// TIA Portal V20 export
DATA_BLOCK "EmData"   // DB92
// stored: Access Published, MemoryReserve 100, Namespace Unit1
   VAR
      anodeElectrode : DInt;
      cathodeElectrode : DInt;
      currentTotalElectrode : DInt;
      targetTotalElectrode : DInt := 39;
      oldTotalElectrode : DInt;
      remainValue : DInt;   // Return reminder of divison.
      cpm : DInt := 80;
      homing : Bool;
      ReelCutStackCellCount : LReal;
      PartData : Struct
         EM4 : "LER_typePartDataEm4";
         EM5 : "LER_typePartDataEm5";
         EM6 : "LER_typePartDataEm6";
         EM7 : "LER_typePartDataEm7";
         clearPartData : "LER_typePartData";
         clearTableBuffer : Array[0..59] of "LER_typeUnitData";
      END_STRUCT;
      calculateResult : Struct
         sepaClampCutterAxisX { S7_SetPoint := 'True'} : "LBC_typeAxis64PosConfiguration";
         sepaClampCutterAxisZ { S7_SetPoint := 'True'} : "LBC_typeAxis64PosConfiguration";
         sepaGripperAxisX { S7_SetPoint := 'True'} : "LBC_typeAxis64PosConfiguration";
         pusherAxisZ { S7_SetPoint := 'True'} : "LBC_typeAxis64PosConfiguration";
      END_STRUCT;
      RunOutModeControl : Struct   // Run Out Mode Start
         RunOutStart : Bool;
         RunOutComplete : Bool;
      END_STRUCT;
      UnitRecipe : Struct
         size : "LER.Size";
         SepaThickness { S7_SetPoint := 'True'} : LReal := 0.25;
         JellyRollWidth : LReal;
         StackCount : DInt := 39;
         DancerRegulator : LReal;
         AutoSpliceRemainingLength : LReal;
         TotalSepaWebLenth : LReal;
      END_STRUCT;
   END_VAR
   VAR RETAIN
      DataBit : Struct
         AnodePnP1 : Bool;
         AnodePnP2 : Bool;
         AnodeTable : Bool;
         CathodePnP1 : Bool;
         CathodePnP2 : Bool;
         CathodeTable : Bool;
      END_STRUCT;
   END_VAR
   VAR
      sepaCleanData : Struct
         currentTotalSepa : DInt;
         targetTotalSepa : DInt;
         oldTotalSepa : DInt;
      END_STRUCT;
   END_VAR
BEGIN
   UnitRecipe.size.Anode.thickness := 0.5;
   UnitRecipe.size.Anode.length := 200.0;
   UnitRecipe.size.Cathode.thickness := 0.5;
   UnitRecipe.size.Cathode.length := 200.0;
END_DATA_BLOCK
